PROGRAM MAIN
VAR
END_VAR

//prg_jafunctie();
//prg_TweeSignalen();
//prg_Reactorvat();
//prg_Opslagvat();
//PRG_OpslagFoutDetectie();
//prg_Alarmbewaking();
//prg_Teleruptorschakeling();
//prg_MotorMetDrukknop();
//prg_TweePompen();
//prg_DriePompen();
prg_Verschalingmetfunctie();

END_PROGRAM

(* stored: Version 1.1.0.1, ProductVersion 3.1.4024.15
   POU MAIN: Id {06c787c3-cfd1-4301-ab7e-6520ebb35bc3}, SpecialFunc None *)
